// TIA Portal V18 export
TYPE "RCS_SysManual_V1"
// stored: IsFailsafeCompliant false
   STRUCT
      Mode : Bool;   // Sation in Manual Mode (bit tag)
      BtnCanActivate : Bool;   // Manual Button Can be Activated
   END_STRUCT;
END_TYPE
